// TwinCAT 3 PLC project TrafficLightAppPLC
// ProgramVersion: 3.1.4024.0
// libraries:
//   Tc2_Standard, * (Beckhoff Automation GmbH)
//   Tc2_System, * (Beckhoff Automation GmbH)
//   Tc3_Module, * (Beckhoff Automation GmbH)
//   TrafficControlLib, * (TrafficLightProject AG)
// project tree:
//   / PlcTask.TcTTO
//   POUs/ MAIN.TcPOU
// real-time tasks:
//   TASK PlcTask: cycle T#10ms, priority 20, ADS port 350
//   TASK PlcTask1: cycle T#10ms, priority 21, ADS port 351

CONFIGURATION TrafficLightAppPLC
    RESOURCE PLC ON TwinCAT3
        TASK PlcTask(INTERVAL := T#10ms, PRIORITY := 20);
        PROGRAM MAIN WITH PlcTask : MAIN;
    END_RESOURCE
END_CONFIGURATION

// ---- POUs/MAIN.TcPOU
PROGRAM MAIN
VAR
	fbIntersection : FB_Intersection;
    tonAdvance     : TON;                        // timer between phase advances
    PHASE_TIME     : TIME := T#5S;               // how long each phase lasts
	bManualAdvance : BOOL := FALSE;			     // HMI button
END_VAR

// Auto-advance on timer
tonAdvance(IN := NOT tonAdvance.Q, PT := PHASE_TIME);
IF (tonAdvance.Q) THEN
    fbIntersection.Advance();
END_IF

// Manual advance from HMI (edge-detected inside the intersection)
fbIntersection.Update(bManualStepRequest := bManualAdvance);

END_PROGRAM
